ORGANIZATION_BLOCK PRINCIPAL:OB1
TITLE=COMENTARIOS DEL PROGRAMA
BEGIN
Network 1
LD     I1.0
O      Q0.0
AN     I0.2
=      Q0.0
Network 2
LD     I0.0
O      I0.1
O      I0.2
=      Q0.1
Network 3
LDN    I0.0
A      I0.1
A      I0.2
O      Q0.3
AN     T37
AN     Q0.4
=      Q0.3
Network 4
LD     I0.0
A      I0.2
O      Q0.4
AN     T37
AN     Q0.3
=      Q0.4
Network 5
LD     Q0.3
O      Q0.4
TON    T37, 250
END_ORGANIZATION_BLOCK
SUBROUTINE_BLOCK SBR_0:SBR0
TITLE=COMENTARIOS DE LA SUBRUTINA
BEGIN
Network 1 // Título de segmento
// Comentario de segmento
END_SUBROUTINE_BLOCK
INTERRUPT_BLOCK INT_0:INT0
TITLE=COMENTARIOS DE LA RUTINA DE INTERRUPCIÓN
BEGIN
Network 1 // Título de segmento
// Comentario de segmento
END_INTERRUPT_BLOCK
